// LS Electric XG5000 project: 과년65_3
// PLC NewPLC
// module base 0 slot 0: 입출력 모듈:XBC-DR20S (DC 24V 입력 12점, 릴레이 출력 8점)

PROGRAM NewProgram (task: 스캔 프로그램)

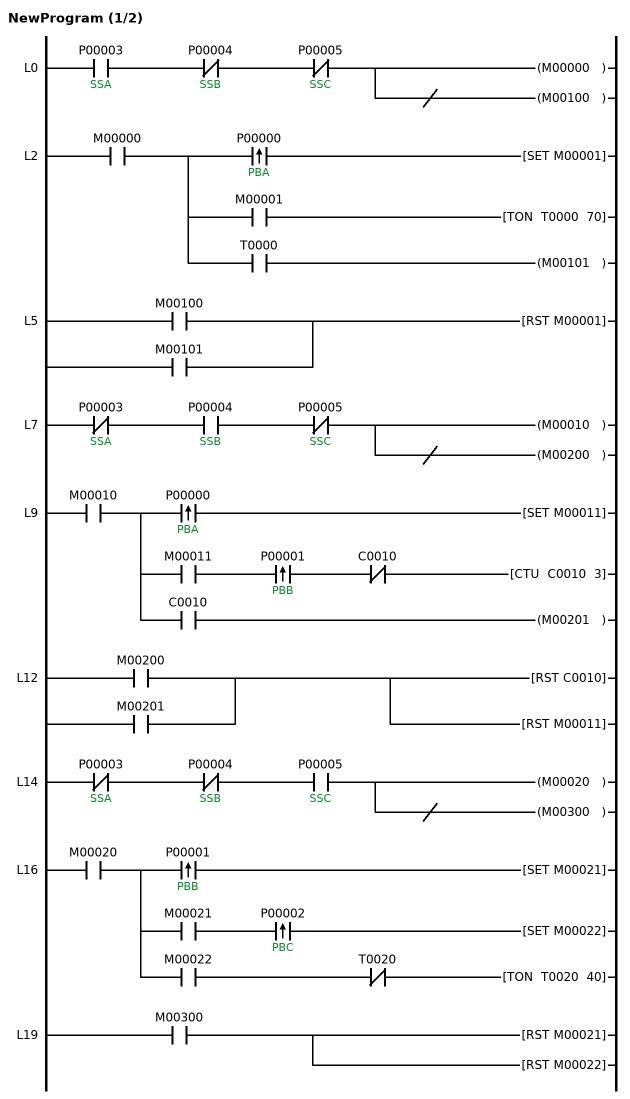
; L0
LOAD      P00003	// SSA
AND NOT   P00004	// SSB
AND NOT   P00005	// SSC
OUT       M00000
NOT
OUT       M00100
; L2
LOAD      M00000
MPUSH
ANDP      P00000	// PBA
SET       M00001
MLOAD
AND       M00001
TON       T0000 70
MPOP
AND       T0000
OUT       M00101
; L5
LOAD      M00100
OR        M00101
RST       M00001
; L7
LOAD NOT  P00003	// SSA
AND       P00004	// SSB
AND NOT   P00005	// SSC
OUT       M00010
NOT
OUT       M00200
; L9
LOAD      M00010
MPUSH
ANDP      P00000	// PBA
SET       M00011
MLOAD
AND       M00011
ANDP      P00001	// PBB
AND NOT   C0010
CTU       C0010 3
MPOP
AND       C0010
OUT       M00201
; L12
LOAD      M00200
OR        M00201
RST       C0010
RST       M00011
; L14
LOAD NOT  P00003	// SSA
AND NOT   P00004	// SSB
AND       P00005	// SSC
OUT       M00020
NOT
OUT       M00300
; L16
LOAD      M00020
MPUSH
ANDP      P00001	// PBB
SET       M00021
MLOAD
AND       M00021
ANDP      P00002	// PBC
SET       M00022
MPOP
AND       M00022
AND NOT   T0020
TON       T0020 40
; L19
LOAD      M00300
RST       M00021
RST       M00022

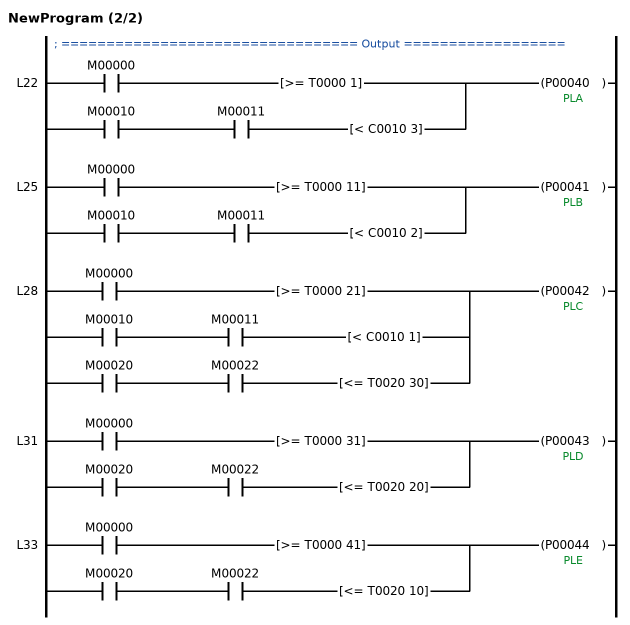
// ================================= Output ==================
; L22
LOAD      M00000
AND>=     T0000 1
LOAD      M00010
AND       M00011
AND<      C0010 3
OR LOAD
OUT       P00040	// PLA
; L25
LOAD      M00000
AND>=     T0000 11
LOAD      M00010
AND       M00011
AND<      C0010 2
OR LOAD
OUT       P00041	// PLB
; L28
LOAD      M00000
AND>=     T0000 21
LOAD      M00010
AND       M00011
AND<      C0010 1
OR LOAD
LOAD      M00020
AND       M00022
AND<=     T0020 30
OR LOAD
OUT       P00042	// PLC
; L31
LOAD      M00000
AND>=     T0000 31
LOAD      M00020
AND       M00022
AND<=     T0020 20
OR LOAD
OUT       P00043	// PLD
; L33
LOAD      M00000
AND>=     T0000 41
LOAD      M00020
AND       M00022
AND<=     T0020 10
OR LOAD
OUT       P00044	// PLE